(* IEC 61131-3 sources: Std_PalletMover/Class/I_Lift, 1 file *)

(* ---- I_Lift.st ---- *)
(*!
<Class
	Name               = "I_Lift"
	Revision           = "0.0"
	RealtimeTask       = "false"
	CyclicTask         = "false"
	BackgroundTask     = "false"
	Sigmatek           = "false"
	OSInterface        = "false"
	HighPriority       = "false"
	Automatic          = "false"
	UpdateMode         = "Prescan"
	SharedCommandTable = "true"
	Objectsize         = "(630,360)">
	<Channels>
		<Server Name="ActualHeight" Visualized="false" Initialize="false" WriteProtected="true" Retentive="false"/>
		<Server Name="ClassSvr" Visualized="false" Initialize="false" WriteProtected="true" Retentive="false"/>
		<Server Name="SetHeight" Visualized="false" Initialize="false" WriteProtected="true" Retentive="false"/>
		<Server Name="SetSpeed" Visualized="false" Initialize="false" WriteProtected="true" Retentive="false"/>
		<Server Name="State" Visualized="false" Initialize="false" WriteProtected="true" Retentive="false"/>
	</Channels>
</Class>
*)
I_Lift : CLASS
	TYPE
	  LiftState : BDINT  //! <Type Public="true" Name="LiftState"/>
	  [
	    1 OnTarget,
	    2 MovingUp,
	    3 MovingDown,
	    4 Bit4,
	    5 Bit5,
	    6 Bit6,
	    7 Bit7,
	    8 Bit8,
	    9 Bit9,
	    10 Bit10,
	    11 Bit11,
	    12 Bit12,
	    13 Bit13,
	    14 Bit14,
	    15 Bit15,
	    16 Bit16,
	    17 Bit17,
	    18 Bit18,
	    19 Bit19,
	    20 Bit20,
	    21 Bit21,
	    22 Bit22,
	    23 Bit23,
	    24 Bit24,
	    25 Bit25,
	    26 Bit26,
	    27 Bit27,
	    28 Bit28,
	    29 Bit29,
	    30 Bit30,
	    31 ReadyToUse,
	    32 InError,
	  ];
	END_TYPE
  //Servers:
	ClassSvr 	: SvrChCmd_DINT;
	ActualHeight 	: SvrCh_DINT;
	SetHeight 	: SvrCh_DINT;
	SetSpeed 	: SvrCh_DINT;
	State 	: SvrCh_LiftState_PTofCls_I_Lift;
  //Clients:
  //Variables:
  //Functions:
  //Tables:
	FUNCTION @STD
		VAR_OUTPUT
			ret_code	: CONFSTATES;
		END_VAR;
	FUNCTION GLOBAL TAB @CT_;
END_CLASS;
